// TwinCAT 3 PLC project Simulation
// ProgramVersion: 3.1.4024.0
// libraries:
//   Tc2_Standard, * (Beckhoff Automation GmbH)
//   Tc2_System, * (Beckhoff Automation GmbH)
//   Tc3_Module, * (Beckhoff Automation GmbH)
// project tree:
//   / PlcTask.TcTTO
//   POUs/ FB_CurtainResp.TcPOU, MAIN.TcPOU
// (motion and I/O tree: see PLC project plc)
// real-time tasks:
//   TASK PlcTask: cycle T#10ms, priority 20, ADS port 350
//   TASK PlcTask1: cycle T#10ms, priority 21, ADS port 351

CONFIGURATION Simulation
    RESOURCE PLC ON TwinCAT3
        TASK PlcTask(INTERVAL := T#10ms, PRIORITY := 21);
        PROGRAM MAIN WITH PlcTask : MAIN;
    END_RESOURCE
END_CONFIGURATION

// ---- POUs/MAIN.TcPOU
PROGRAM MAIN
VAR
	fbCurtainResp: FB_CurtainResp;
END_VAR


	fbCurtainResp(
	Open:= , 
	Close:= , 
	OpenToCloseTime:= , 
	plcCylTime_mSec:= , 
	AtOpen=> , 
	AtClose=> );

END_PROGRAM

// ---- POUs/FB_CurtainResp.TcPOU
FUNCTION_BLOCK FB_CurtainResp
VAR_INPUT
	Open	 AT%I* : BOOL;
	Close	 AT%I* : BOOL;
	OpenToCloseTime: INT := 10000;		
	plcCylTime_mSec: INT := 10;	
END_VAR
VAR_OUTPUT
	AtOpen	 AT%Q* 	: BOOL;		// Sensor Feedback	
	AtClose	 AT%Q*	: BOOL;		// Sensor Feedback
END_VAR
VAR
	OpenTime: INT;
	rtAtOpen: R_TRIG;
	rtAtClose: R_TRIG;
END_VAR


	rtAtOpen(CLK:= AtOpen, Q=> );
	rtAtClose(CLK:= AtClose, Q=> );

	IF rtAtOpen.Q OR rtAtClose.Q THEN
		;//OpenTime	:=	0;
	END_IF
	
	OpenTime	:=	LIMIT(0 , OpenTime , OpenToCloseTime);

	IF Open AND (NOT Close) THEN
		OpenTime := OpenTime + plcCylTime_mSec;
		AtOpen	:=	FALSE;
		AtClose :=	FALSE;
	END_IF
	IF OpenTime >= OpenToCloseTime THEN
		AtOpen	:=	TRUE;
		AtClose	:=	FALSE;
	END_IF

	IF Close AND (NOT Open) THEN
		OpenTime := (OpenTime - plcCylTime_mSec);
		AtOpen	:=	FALSE;
		AtClose :=	FALSE;
	END_IF
	IF OpenTime <= 0 THEN
		AtOpen	:=	FALSE;
		AtClose :=	TRUE;
	END_IF

END_FUNCTION_BLOCK
